FUNCTION_BLOCK TN_SC_READ_ATTR
VAR
	in_Offset : INT;
END_VAR
VAR_INPUT
	Iin_Y : INT;
	Iin_X : INT;
END_VAR
VAR_OUTPUT
	Oby_ATTR : BYTE;
END_VAR
VAR_IN_OUT
	Xus_TN_SCREEN : us_TN_SCREEN;
END_VAR

(*
version 1.0		10. mai 2010
programmer		ks
tested by		ks

TN_SC_READ_ATTR gibt den Farbcode einer Koordinate vom Bildschirm aus

*)

IF TN_SC_XY_ERROR(Iin_X,Iin_Y) THEN RETURN; END_IF;
in_Offset := (Iin_Y * 80) + Iin_X;
Oby_ATTR := Xus_TN_SCREEN.bya_COLOR[in_Offset]; (* Attribute auslesen *)

(* revision history
ks	10. mai. 2010	rev 1.0
	original version
*)

END_FUNCTION_BLOCK

(* stored: Version 1.1.0.1, ProductVersion 3.1.4022.7
   POU TN_SC_READ_ATTR: Id {5cb9e455-48ac-4d9b-8e84-ed317f8028d4}, SpecialFunc None *)
